FUNCTION_BLOCK PLCControl (* Basic Function Block Type *)
  (* Standard: 61499-2 *)
  (* Version 0.0, 6/17/2016, Andrei, nxtControl GmbH, Template *)
  PACKAGE Main;
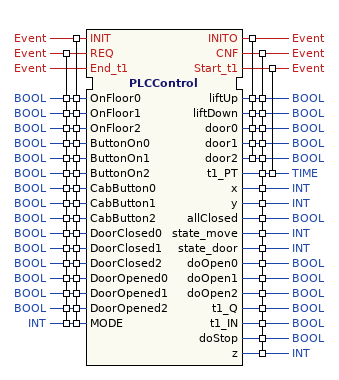
  EVENT_INPUT
    INIT WITH OnFloor0, OnFloor1, OnFloor2, ButtonOn0, ButtonOn1, ButtonOn2, CabButton0, CabButton1, CabButton2, DoorClosed0, DoorClosed1, DoorClosed2, DoorOpened0, DoorOpened1, DoorOpened2, MODE; (* Initialization Request *)
    REQ WITH OnFloor0, OnFloor1, OnFloor2, ButtonOn0, ButtonOn1, ButtonOn2, CabButton0, CabButton1, CabButton2, DoorClosed0, DoorClosed1, DoorClosed2, DoorOpened0, DoorOpened1, DoorOpened2, MODE; (* Normal Execution Request *)
    End_t1;
  END_EVENT
  EVENT_OUTPUT
    INITO WITH liftUp, liftDown, door0, door1, door2; (* Initialization Confirm *)
    CNF WITH liftUp, liftDown, door0, door1, door2, t1_PT, x, y, allClosed, state_move, state_door, doOpen0, doOpen1, doOpen2, t1_Q, t1_IN, doStop, z; (* Execution Confirmation *)
    Start_t1 WITH t1_PT;
  END_EVENT
  VAR_INPUT
    OnFloor0 : BOOL; (* Input event qualifier *)
    OnFloor1 : BOOL;
    OnFloor2 : BOOL;
    ButtonOn0 : BOOL;
    ButtonOn1 : BOOL;
    ButtonOn2 : BOOL;
    CabButton0 : BOOL;
    CabButton1 : BOOL;
    CabButton2 : BOOL;
    DoorClosed0 : BOOL;
    DoorClosed1 : BOOL;
    DoorClosed2 : BOOL;
    DoorOpened0 : BOOL;
    DoorOpened1 : BOOL;
    DoorOpened2 : BOOL;
    MODE : INT;
  END_VAR
  VAR_OUTPUT
    liftUp : BOOL;
    liftDown : BOOL; (* Output event qualifier *)
    door0 : BOOL;
    door1 : BOOL;
    door2 : BOOL;
    t1_PT : TIME;
    x : INT;
    y : INT;
    allClosed : BOOL;
    state_move : INT;
    state_door : INT;
    doOpen0 : BOOL;
    doOpen1 : BOOL;
    doOpen2 : BOOL;
    t1_Q : BOOL;
    t1_IN : BOOL;
    doStop : BOOL;
    z : INT;
  END_VAR
  VAR
    STATE_STOPPED : INT := 0;
    STATE_GOING_UP : INT := 1;
    STATE_GOING_DOWN : INT := 2;
    STATE_CLOSED : INT := 0;
    STATE_OPENING0 : INT := 1;
    STATE_OPENING1 : INT := 2;
    STATE_OPENING2 : INT := 3;
    STATE_OPEN : INT := 4;
    STATE_CLOSING : INT := 5;
  END_VAR
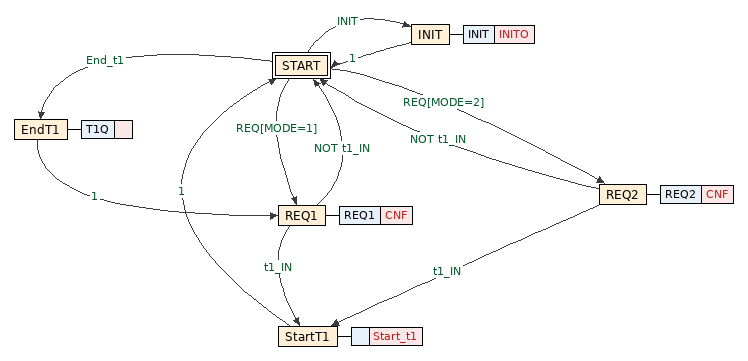
  EC_STATES
    START; (* Initial State *)
    INIT : INIT -> INITO;
    REQ1 : REQ1 -> CNF;
    StartT1 : -> Start_t1;
    EndT1 : T1Q;
    REQ2 : REQ2 -> CNF;
  END_STATES
  EC_TRANSITIONS
    START TO INIT := INIT;
    INIT TO START := 1;
    START TO REQ1 := REQ[MODE=1];
    REQ1 TO StartT1 := t1_IN;
    StartT1 TO START := 1;
    START TO EndT1 := End_t1;
    EndT1 TO REQ1 := 1;
    REQ1 TO START := NOT t1_IN;
    START TO REQ2 := REQ[MODE=2];
    REQ2 TO START := NOT t1_IN;
    REQ2 TO StartT1 := t1_IN;
  END_TRANSITIONS
  ALGORITHM INIT IN ST: (* Initialization algorithm *)
;
t1_IN :=FALSE;
t1_Q  :=FALSE;
state_move := STATE_STOPPED;
state_door := STATE_CLOSED;
  END_ALGORITHM
  ALGORITHM REQ1 IN ST: (* Normally executed algorithm *)
;

allClosed := DoorClosed0 AND DoorClosed1 AND DoorClosed2;



IF ButtonOn0 OR CabButton0 THEN
	x:= 0;
ELSIF ButtonOn1 OR CabButton1 THEN
	x:= 1;
ELSIF ButtonOn2 OR CabButton2 THEN
	x:= 2;
ELSE
	x:=-2;
END_IF;

IF OnFloor0 THEN
	y:= 0;
ELSIF OnFloor1 THEN
	y:=1;
ELSIF OnFloor2 THEN
	y:=2;
ELSE
	y:=-2;
END_IF;

doStop := (y=0 AND (ButtonOn0 OR CabButton0)) OR (y=1 AND (ButtonOn1 OR CabButton1)) OR (y=2 AND (ButtonOn2 OR CabButton2));
doOpen0 := y=0 AND (ButtonOn0 OR CabButton0);
doOpen1 := y=1 AND (ButtonOn1 OR CabButton1);
doOpen2 := y=2 AND (ButtonOn2 OR CabButton2);



IF state_move = STATE_STOPPED THEN
	liftUp := FALSE; liftDown:= FALSE;
	IF allClosed AND x < y AND x >= 0 THEN
		state_move:= STATE_GOING_DOWN;
	ELSIF allClosed AND x > y AND x >= 0 THEN
		state_move:= STATE_GOING_UP;
	END_IF;
ELSIF state_move = STATE_GOING_UP THEN
	liftUp:=TRUE; liftDown:= FALSE;
	IF doStop THEN
		state_move := STATE_STOPPED;
	END_IF;
ELSIF state_move = STATE_GOING_DOWN THEN
	liftDown:= TRUE; liftUp:= FALSE;
	IF doStop THEN
		state_move := STATE_STOPPED;
	END_IF;
END_IF;

IF state_door = STATE_CLOSED THEN
	IF doOpen0 THEN
		state_door := STATE_OPENING0;
	ELSIF doOpen1 THEN
		state_door := STATE_OPENING1;
	ELSIF doOpen2 THEN
		state_door := STATE_OPENING2;
	END_IF;
ELSIF state_door = STATE_OPENING0 THEN
	door0:= TRUE;
	IF DoorOpened0 THEN
		state_door := STATE_OPEN;
	END_IF;
ELSIF state_door = STATE_OPENING1 THEN
	door1:=TRUE;
	IF DoorOpened1 THEN
		state_door := STATE_OPEN;
	END_IF;
ELSIF state_door = STATE_OPENING2 THEN
	door2:=TRUE;
	IF DoorOpened2 THEN
		state_door := STATE_OPEN;
	END_IF;
ELSIF state_door = STATE_OPEN THEN
	t1_IN:=TRUE;
	t1_PT:=T#3S;
	Start_t1:=TRUE;
	IF t1_Q  THEN
		t1_IN:=FALSE;
		End_t1:=TRUE;
		t1_Q := FALSE;
		state_door := STATE_CLOSING;
	END_IF;
ELSIF state_door = STATE_CLOSING THEN
	door0:= FALSE;
	door1:= FALSE;
	door2:= FALSE;
	IF allClosed THEN
		state_door := STATE_CLOSED;
	END_IF;
END_IF;
  END_ALGORITHM
  ALGORITHM T1Q IN ST:
t1_Q:=TRUE;
  END_ALGORITHM
  ALGORITHM REQ2 IN ST:
;
allClosed := DoorClosed0 AND DoorClosed1 AND DoorClosed2;

IF CabButton0 THEN
	z:= 0;
ELSIF CabButton1 THEN
	z:= 1;
ELSIF CabButton2 THEN
	z:= 2;
ELSE
	z:=-2;
END_IF;

IF ButtonOn0 THEN
	x:= 0;
ELSIF ButtonOn1 THEN
	x:= 1;
ELSIF ButtonOn2 THEN
	x:= 2;
ELSE
	x:=-2;
END_IF;

IF OnFloor0 THEN
	y:= 0;
ELSIF OnFloor1 THEN
	y:=1;
ELSIF OnFloor2 THEN
	y:=2;
ELSE
	y:=-2;
END_IF;

doStop := (y=0 AND (ButtonOn0 OR CabButton0)) OR (y=1 AND (ButtonOn1 OR CabButton1)) OR (y=2 AND (ButtonOn2 OR CabButton2));
doOpen0 := y=0 AND (ButtonOn0 OR CabButton0);
doOpen1 := y=1 AND (ButtonOn1 OR CabButton1);
doOpen2 := y=2 AND (ButtonOn2 OR CabButton2);




IF state_move = STATE_STOPPED THEN
	liftUp := FALSE; liftDown:= FALSE;
	IF allClosed AND z < y AND z >= 0 THEN
	state_move:= STATE_GOING_DOWN;
	ELSIF allClosed AND z > y AND z >= 0 THEN
	state_move:= STATE_GOING_UP;
	ELSIF allClosed AND x < y AND x >= 0 THEN
		state_move:= STATE_GOING_DOWN;
	ELSIF allClosed AND x > y AND x >= 0 THEN
		state_move:= STATE_GOING_UP;
	END_IF;
ELSIF state_move = STATE_GOING_UP THEN
	liftUp:=TRUE; liftDown:= FALSE;
	IF doStop THEN
		state_move := STATE_STOPPED;
	END_IF;
ELSIF state_move = STATE_GOING_DOWN THEN
	liftDown:= TRUE; liftUp:= FALSE;
	IF doStop THEN
		state_move := STATE_STOPPED;
	END_IF;
END_IF;

IF state_door = STATE_CLOSED THEN
	IF doOpen0 THEN
		state_door := STATE_OPENING0;
	ELSIF doOpen1 THEN
		state_door := STATE_OPENING1;
	ELSIF doOpen2 THEN
		state_door := STATE_OPENING2;
	END_IF;
ELSIF state_door = STATE_OPENING0 THEN
	door0:= TRUE;
	IF DoorOpened0 THEN
		state_door := STATE_OPEN;
	END_IF;
ELSIF state_door = STATE_OPENING1 THEN
	door1:=TRUE;
	IF DoorOpened1 THEN
		state_door := STATE_OPEN;
	END_IF;
ELSIF state_door = STATE_OPENING2 THEN
	door2:=TRUE;
	IF DoorOpened2 THEN
		state_door := STATE_OPEN;
	END_IF;
ELSIF state_door = STATE_OPEN THEN
	t1_IN:=TRUE;
	t1_PT:=T#3S;
	Start_t1:=TRUE;
	IF t1_Q  THEN
		t1_IN:=FALSE;
		End_t1:=TRUE;
		t1_Q := FALSE;
		state_door := STATE_CLOSING;
	END_IF;
ELSIF state_door = STATE_CLOSING THEN
	door0:= FALSE;
	door1:= FALSE;
	door2:= FALSE;
	IF allClosed THEN
		state_door := STATE_CLOSED;
	END_IF;
END_IF;
  END_ALGORITHM
END_FUNCTION_BLOCK
